(* CoDeSys 2.3 export: ERROR.EXP *)

(* Data type in STRUCT *)
TYPE Error :
STRUCT
	err_code: UINT;
	par1: UINT;
	par2: UINT;
END_STRUCT
END_TYPE
